FUNCTION_BLOCK T_CyclicLogicHasBeenCalledTrue EXTENDS T_UnitTestBase
VAR
  list : T_ComponentsCollection(10);
  newComponent, newComponent2 : T_Component; 
  actual1, actual2 : BOOL;
END_VAR

// Arrange
list.AddComponent(newComponent);
list.AddComponent(newComponent2);

//Act
list.CyclicLogic();

//Assert
actual1 := newComponent.cyclicHasBeenCalled;
actual2 := newComponent2.cyclicHasBeenCalled;

assertion.AssertEquals_BOOL(TRUE, actual1, 'actual1 := newComponent.cyclicHasBeenCalled;');
assertion.AssertEquals_BOOL(TRUE, actual2, 'actual2 := newComponent2.cyclicHasBeenCalled');
TestFinished();

END_FUNCTION_BLOCK

(* stored: Version 1.1.0.1, ProductVersion 3.1.4024.12
   POU T_CyclicLogicHasBeenCalledTrue: Id {8d4fac65-8965-408a-b985-1027762b7472}, SpecialFunc None *)
